Fanuc KAREL source: WeldTriangleWeave.kl

PROGRAM WELDTRIANGLEWEAVE
%NOLOCKGROUP
%NOPAUSE = ERROR + COMMAND + TPENABLE
%COMMENT = 'Triangle weave placeholder'

BEGIN
  WRITE('WELDTRIANGLEWEAVE START', CR)
  WRITE('Implement triangle weave motion here.', CR)
END WELDTRIANGLEWEAVE
